(* IEC 61131-3 sources: fbd-complexity-tool/src/test/resources/test1/build, 2 files *)

(* ---- generated_plc.st ---- *)
TYPE
  CalType : REAL := 5.0;
END_TYPE

FUNCTION_BLOCK Volume
  VAR_INPUT
    BalControl : SINT;
    VolControl : SINT;
    ModelType : BOOL;
  END_VAR
  VAR_OUTPUT
    RightAmplif : REAL;
    LeftAmplif : REAL;
    LED : BOOL;
  END_VAR
  VAR_IN_OUT
    Critical : BOOL;
  END_VAR
  VAR
    MaxVolume : REAL := 26.0;
    HeatTime : TON;
    Overdrive : BOOL;
  END_VAR

  HeatTime();
END_FUNCTION_BLOCK

FUNCTION Norm : BOOL
  VAR_INPUT
    BIK : SINT;
    LCtrlK : SINT;
    MType : BOOL;
  END_VAR
  VAR
    Calib : CalType;
  END_VAR
  VAR_OUTPUT
    Norm : REAL;
  END_VAR
  VAR
    SINT_TO_REAL1_OUT : REAL;
    SEL6_OUT : REAL;
    SINT_TO_REAL9_OUT : REAL;
    ADD7_OUT : BOOL;
  END_VAR

  SINT_TO_REAL1_OUT := SINT_TO_REAL(BIK);
  SEL6_OUT := SEL(MType);
  SINT_TO_REAL9_OUT := SINT_TO_REAL(LCtrlK);
  ADD7_OUT := ADD(SINT_TO_REAL1_OUT, SEL6_OUT, Calib, SINT_TO_REAL9_OUT);
  Norm := ADD7_OUT;
END_FUNCTION

CONFIGURATION config

  RESOURCE resource0 ON PLC
  END_RESOURCE
END_CONFIGURATION

(* ---- plc.st ---- *)
TYPE
  LOGLEVEL : (CRITICAL, WARNING, INFO, DEBUG) := INFO;
END_TYPE

FUNCTION_BLOCK LOGGER
  VAR_INPUT
    TRIG : BOOL;
    MSG : STRING;
    LEVEL : LOGLEVEL := INFO;
  END_VAR
  VAR
    TRIG0 : BOOL;
  END_VAR

  IF TRIG AND NOT TRIG0 THEN
  {{
   LogMessage(GetFbVar(LEVEL),(char*)GetFbVar(MSG, .body),GetFbVar(MSG, .len));
  }}
  END_IF;
  TRIG0:=TRIG;
END_FUNCTION_BLOCK

FUNCTION_BLOCK python_eval
  VAR_INPUT
    TRIG : BOOL;
    CODE : STRING;
  END_VAR
  VAR_OUTPUT
    ACK : BOOL;
    RESULT : STRING;
  END_VAR
  VAR
    STATE : DWORD;
    BUFFER : STRING;
    PREBUFFER : STRING;
    TRIGM1 : BOOL;
    TRIGGED : BOOL;
  END_VAR

  {extern void __PythonEvalFB(int, PYTHON_EVAL*);__PythonEvalFB(0, data__);}
END_FUNCTION_BLOCK

FUNCTION_BLOCK python_poll
  VAR_INPUT
    TRIG : BOOL;
    CODE : STRING;
  END_VAR
  VAR_OUTPUT
    ACK : BOOL;
    RESULT : STRING;
  END_VAR
  VAR
    STATE : DWORD;
    BUFFER : STRING;
    PREBUFFER : STRING;
    TRIGM1 : BOOL;
    TRIGGED : BOOL;
  END_VAR

  {extern void __PythonEvalFB(int, PYTHON_EVAL*);__PythonEvalFB(1,(PYTHON_EVAL*)(void*)data__);}
END_FUNCTION_BLOCK

FUNCTION_BLOCK python_gear
  VAR_INPUT
    N : UINT;
    TRIG : BOOL;
    CODE : STRING;
  END_VAR
  VAR_OUTPUT
    ACK : BOOL;
    RESULT : STRING;
  END_VAR
  VAR
    py_eval : python_eval;
    COUNTER : UINT;
    ADD10_OUT : UINT;
    EQ13_OUT : BOOL;
    SEL15_OUT : UINT;
    AND7_OUT : BOOL;
  END_VAR

  ADD10_OUT := ADD(COUNTER, 1);
  EQ13_OUT := EQ(N, ADD10_OUT);
  SEL15_OUT := SEL(EQ13_OUT, ADD10_OUT, 0);
  COUNTER := SEL15_OUT;
  AND7_OUT := AND(EQ13_OUT, TRIG);
  py_eval(TRIG := AND7_OUT, CODE := CODE);
  ACK := py_eval.ACK;
  RESULT := py_eval.RESULT;
END_FUNCTION_BLOCK

FUNCTION_BLOCK GetBoolString
  VAR_INPUT
    VALUE : BOOL;
  END_VAR
  VAR_OUTPUT
    CODE : STRING;
  END_VAR

  IF VALUE THEN
    CODE := 'True';
  ELSE
    CODE := 'False';
  END_IF;
END_FUNCTION_BLOCK

FUNCTION_BLOCK Button
  VAR
    ID : STRING;
  END_VAR
  VAR_INPUT
    back_id : STRING;
    sele_id : STRING;
    toggle : BOOL;
    set_state : BOOL;
    state_in : BOOL;
  END_VAR
  VAR_OUTPUT
    state_out : BOOL;
  END_VAR
  VAR
    init_Command : python_eval;
    GetButtonState : GetBoolString;
    setstate_Command : python_eval;
    getstate_Command : python_poll;
    GetButtonToggle : GetBoolString;
    CONCAT2_OUT : STRING;
    CONCAT22_OUT : STRING;
    STRING_TO_INT25_OUT : INT;
    INT_TO_BOOL26_OUT : BOOL;
    AND31_OUT : BOOL;
    CONCAT7_OUT : STRING;
  END_VAR

  GetButtonToggle(VALUE := toggle);
  CONCAT2_OUT := CONCAT('createSVGUIControl("button",back_id="', back_id, '",sele_id="', sele_id, '",toggle=', GetButtonToggle.CODE, ',active=True)');
  init_Command(TRIG := BOOL#1, CODE := CONCAT2_OUT);
  ID := init_Command.RESULT;
  CONCAT22_OUT := CONCAT('int(getAttr(', ID, ',"state",False))');
  getstate_Command(TRIG := init_Command.ACK, CODE := CONCAT22_OUT);
  STRING_TO_INT25_OUT := STRING_TO_INT(getstate_Command.RESULT);
  INT_TO_BOOL26_OUT := INT_TO_BOOL(STRING_TO_INT25_OUT);
  state_out := INT_TO_BOOL26_OUT;
  AND31_OUT := AND(init_Command.ACK, set_state);
  GetButtonState(VALUE := state_in);
  CONCAT7_OUT := CONCAT('setAttr(', ID, ',"state",', GetButtonState.CODE, ')');
  setstate_Command(TRIG := AND31_OUT, CODE := CONCAT7_OUT);
END_FUNCTION_BLOCK

FUNCTION_BLOCK Led
  VAR
    ID : STRING;
  END_VAR
  VAR_INPUT
    back_id : STRING;
    sele_id : STRING;
    state_in : BOOL;
  END_VAR
  VAR
    init_Command : python_eval;
    setstate_Command : python_poll;
    GetLedState : GetBoolString;
    CONCAT2_OUT : STRING;
    CONCAT7_OUT : STRING;
  END_VAR

  CONCAT2_OUT := CONCAT('createSVGUIControl("button",back_id="', back_id, '",sele_id="', sele_id, '",toggle=True,active=False)');
  init_Command(TRIG := BOOL#1, CODE := CONCAT2_OUT);
  ID := init_Command.RESULT;
  GetLedState(VALUE := state_in);
  CONCAT7_OUT := CONCAT('setAttr(', ID, ',"state",', GetLedState.CODE, ')');
  setstate_Command(TRIG := init_Command.ACK, CODE := CONCAT7_OUT);
END_FUNCTION_BLOCK

FUNCTION_BLOCK TextCtrl
  VAR
    ID : STRING;
  END_VAR
  VAR_INPUT
    back_id : STRING;
    set_text : BOOL;
    text : STRING;
  END_VAR
  VAR
    SVGUI_TEXTCTRL : python_eval;
    setstate_Command : python_eval;
    CONCAT1_OUT : STRING;
    AND31_OUT : BOOL;
    CONCAT12_OUT : STRING;
  END_VAR

  CONCAT1_OUT := CONCAT('createSVGUIControl("textControl", back_id="', back_id, '")');
  SVGUI_TEXTCTRL(TRIG := BOOL#1, CODE := CONCAT1_OUT);
  ID := SVGUI_TEXTCTRL.RESULT;
  AND31_OUT := AND(SVGUI_TEXTCTRL.ACK, set_text);
  CONCAT12_OUT := CONCAT('setAttr(', ID, ',"text","', text, '")');
  setstate_Command(TRIG := AND31_OUT, CODE := CONCAT12_OUT);
END_FUNCTION_BLOCK

TYPE
  CalType : REAL := 5.0;
END_TYPE

FUNCTION_BLOCK Volume
  VAR_INPUT
    BalControl : SINT;
    VolControl : SINT;
    ModelType : BOOL;
  END_VAR
  VAR_OUTPUT
    RightAmplif : REAL;
    LeftAmplif : REAL;
    LED : BOOL;
  END_VAR
  VAR_IN_OUT
    Critical : BOOL;
  END_VAR
  VAR
    MaxVolume : REAL := 26.0;
    HeatTime : TON;
    Overdrive : BOOL;
  END_VAR

  HeatTime();
END_FUNCTION_BLOCK

FUNCTION Norm : BOOL
  VAR_INPUT
    BIK : SINT;
    LCtrlK : SINT;
    MType : BOOL;
  END_VAR
  VAR
    Calib : CalType;
  END_VAR
  VAR_OUTPUT
    Norm : REAL;
  END_VAR
  VAR
    SINT_TO_REAL1_OUT : REAL;
    SEL6_OUT : REAL;
    SINT_TO_REAL9_OUT : REAL;
    ADD7_OUT : BOOL;
  END_VAR

  SINT_TO_REAL1_OUT := SINT_TO_REAL(BIK);
  SEL6_OUT := SEL(MType);
  SINT_TO_REAL9_OUT := SINT_TO_REAL(LCtrlK);
  ADD7_OUT := ADD(SINT_TO_REAL1_OUT, SEL6_OUT, Calib, SINT_TO_REAL9_OUT);
  Norm := ADD7_OUT;
END_FUNCTION

CONFIGURATION config

  RESOURCE resource0 ON PLC
  END_RESOURCE
END_CONFIGURATION
